TYPE Heating_Ctx_Io_In :
STRUCT
	bPumpOverload	: BOOL;
	bBurnerOverload	: BOOL;
	
	rBoilerTemp		: LREAL;
	rBoilerPressure	: LREAL;
END_STRUCT
END_TYPE

(* stored: Version 1.1.0.1
   DUT Heating_Ctx_Io_In: Id {f9ff3c65-e6c4-4ead-ae9e-44e73a199f11} *)
